(* IEC 61131-3 sources: SIMERLIFT/LOGICAD/SIMERLIFT/src_FBD/BCU, 6 files *)

(* ---- BatteryTypes.iecst ---- *)
TYPE
    BATTSTATE : USINT( STANDBY := 101,
    				  STARTUP := 102,
    				  PRECHARGE := 103,
    	              DISCHARGE := 104,
                      CHARGE := 105,
                      SHUTDOWN := 106,
                      FAULT := 107,
                      CHARGECOMPLETE := 108,
                      DISCHARGECOMPLETE := 109,
                      PRECHARGE4charge := 110);
END_TYPE

(* ---- ampMaxTempDis.iecst ---- *)
FUNCTION_BLOCK ampMultTempDis {
    width := 200;
  }

VAR_INPUT
temp:REAL;
END_VAR

VAR_OUTPUT
mult : REAL;
END_VAR

VAR
rstTimer:TON;
timeout:BOOL;
lastMult:REAL;
instantMult:REAL;
END_VAR

IF temp<-30 THEN
	mult:=0;
	instantMult:=0;
ELSIF temp<-25  THEN
	instantMult:=0.11;
ELSIF temp<-20  THEN
	instantMult:=0.15;
ELSIF temp<-15  THEN
	instantMult:=0.2;
ELSIF temp<-10  THEN
	instantMult:=0.25;
ELSIF temp<-5  THEN
	instantMult:=0.3;
ELSIF temp<0  THEN
	instantMult:=0.4;
ELSIF temp<5  THEN
	instantMult:=0.5;
ELSIF temp<10  THEN
	instantMult:=0.7;
ELSIF temp<50  THEN
	instantMult:=1;
ELSIF temp<55  THEN
	instantMult:=0.4;
ELSIF temp<56  THEN
	instantMult:=0.2;
ELSE
	mult:=0;
	instantMult:=0;
END_IF;

rstTimer(IN:=instantMult=lastMult, PT:=T#10s, Q=>timeout);

lastMult:=instantMult;

IF timeout THEN
	mult:=instantMult;
END_IF;

END_FUNCTION_BLOCK

(* ---- Arr2Val.iecst ---- *)
FUNCTION_BLOCK ARR2VAL  {
    width := 200;
  }

VAR_INPUT
	MaxBMU:USINT;
    indx:USINT;
	Map:ARRAY[0..15] OF USINT;
	CellCounter:USINT;
END_VAR

VAR_OUTPUT
	numofCell : UINT;
	Reset:BOOL;
END_VAR

Reset:=FALSE;
numofCell:=Map[indx];

IF (NOT Reset) AND (indx = MaxBMU - 1) AND (CellCounter = Map[indx]) THEN
    Reset := TRUE;
END_IF;

END_FUNCTION_BLOCK

(* ---- BCU_ID.iecfbd ---- *)
FUNCTION_BLOCK BCU_ID
  {
    height := 138;
    width := 290;
  }

  VAR
    TON1 : TON;
  END_VAR
  VAR_INPUT
    ADDR_BIT0 : BOOL;
    ADDR_BIT1 : BOOL;
    ADDR_BIT2 : BOOL;
  END_VAR
  VAR_OUTPUT
    PACK_ID : USINT;
    CAN_ID_10 : UDINT;
    CAN_ID_11 : UDINT;
    CAN_ID_12 : UDINT;
    CAN_ID_13 : UDINT;
    CAN_ID_14 : UDINT;
    CAN_ID_15 : UDINT;
    CAN_ID_16 : UDINT;
  END_VAR

  (*

    // Network 1:
    SEL(G := ADDR_BIT0, IN0 := 16#00, IN1 := 16#01, SEL => @C(10).SEL);
    SEL(G := ADDR_BIT1, IN0 := 16#00, IN1 := 16#02, SEL => @C(9).SEL);
    SEL(G := ADDR_BIT2, IN0 := 16#00, IN1 := 16#04, SEL => @C(11).SEL);
    ADD(IN1 := @C(10).SEL, IN2 := @C(9).SEL, IN3 := @C(11).SEL, ADD => PACK_ID);

    // Network 2:
    TON1(IN := 1, PT := T#1s);
    TO_UDINT(IN := TON1.Q, TO_UDINT => @C(36).TO_UDINT);
    ADD(IN1 := 16#18FF10F0, IN2 := PACK_ID, ADD => @C(26).ADD);
    MUL(IN1 := @C(36).TO_UDINT, IN2 := @C(26).ADD, MUL => CAN_ID_10);
    ADD(IN1 := 16#18FF11F0, IN2 := PACK_ID, ADD => @C(30).ADD);
    MUL(IN1 := @C(36).TO_UDINT, IN2 := @C(30).ADD, MUL => CAN_ID_11);
    ADD(IN1 := 16#18FF12F0, IN2 := PACK_ID, ADD => @C(38).ADD);
    MUL(IN1 := @C(36).TO_UDINT, IN2 := @C(38).ADD, MUL => CAN_ID_12);
    ADD(IN1 := 16#18FF13F0, IN2 := PACK_ID, ADD => @C(54).ADD);
    MUL(IN1 := @C(36).TO_UDINT, IN2 := @C(54).ADD, MUL => CAN_ID_13);
    ADD(IN1 := 16#18FF14F0, IN2 := PACK_ID, ADD => @C(25).ADD);
    MUL(IN1 := @C(36).TO_UDINT, IN2 := @C(25).ADD, MUL => CAN_ID_14);
    ADD(IN1 := 16#18FF15F0, IN2 := PACK_ID, ADD => @C(39).ADD);
    MUL(IN1 := @C(36).TO_UDINT, IN2 := @C(39).ADD, MUL => CAN_ID_15);
    ADD(IN1 := 16#18FF16F0, IN2 := PACK_ID, ADD => @C(67).ADD);
    MUL(IN1 := @C(36).TO_UDINT, IN2 := @C(67).ADD, MUL => CAN_ID_16);

  *)

  @VF(4) : @E(16#01), @R(330.0, 120.0, 90.0, 19.0), USINT;
  @C(7) : @F(ADD), @R(660.0, 120.0, 40.0, 58.0), USINT, @I(@N(IN1), @L(9.5)), @I(@N(IN2), @L(29.5)), @I(@N(IN3), @L(49.5)), @O(@N(ADD), @R(9.5));
  @C(10) : @F(SEL), @R(470.0, 80.0, 120.0, 58.0), USINT, @I(@N(G), @L(9.5)), @I(@N(IN0), @L(29.5)), @I(@N(IN1), @L(49.5)), @O(@N(SEL), @R(9.5));
  @C(9) : @F(SEL), @R(470.0, 140.0, 120.0, 58.0), USINT, @I(@N(G), @L(9.5)), @I(@N(IN0), @L(29.5)), @I(@N(IN1), @L(49.5)), @O(@N(SEL), @R(9.5));
  @C(11) : @F(SEL), @R(470.0, 200.0, 120.0, 58.0), USINT, @I(@N(G), @L(9.5)), @I(@N(IN0), @L(29.5)), @I(@N(IN1), @L(49.5)), @O(@N(SEL), @R(9.5));
  @VF(1) : @E(ADDR_BIT0), @R(90.0, 80.0, 140.0, 19.0);
  @VF(14) : @E(16#00), @R(330.0, 100.0, 90.0, 19.0), USINT;
  @VF(17) : @E(ADDR_BIT1), @R(90.0, 140.0, 140.0, 19.0);
  @VF(19) : @E(16#02), @R(330.0, 180.0, 90.0, 19.0), USINT;
  @VF(21) : @E(16#04), @R(330.0, 240.0, 90.0, 19.0), USINT;
  @VF(5) : @E(ADDR_BIT2), @R(90.0, 200.0, 140.0, 19.0);
  @VF(23) : @E(PACK_ID), @R(790.0, 120.0, 140.0, 19.0);
  @VF(468) : @E(16#18FF10F0), @R(280.0, 330.0, 220.0, 19.0), UDINT;
  @VF(33) : @E(CAN_ID_10), @R(790.0, 310.0, 140.0, 19.0);
  @C(41) : @F(MUL), @R(690.0, 310.0, 40.0, 38.0), UDINT, @I(@N(IN1), @L(9.5)), @I(@N(IN2), @L(29.5)), @O(@N(MUL), @R(9.5));
  @C(36) : @F(TO_UDINT), @R(290.0, 310.0, 120.0, 18.0), BOOL, @I(@N(IN), @L(9.5)), @O(@N(TO_UDINT), @R(9.5));
  @C(43) : @FB(TON1), @R(160.0, 310.0, 100.0, 38.0), @I(@N(IN), @L(9.5)), @I(@N(PT), @L(29.5)), @O(@N(Q), @R(9.5)), @O(@N(ET), @R(29.5));
  @VF(46) : @E(1), @R(70.0, 310.0, 70.0, 19.0), BOOL;
  @VF(48) : @E(T#1s), @R(70.0, 330.0, 70.0, 19.0);
  @C(51) : @F(MUL), @R(690.0, 350.0, 40.0, 38.0), UDINT, @I(@N(IN1), @L(9.5)), @I(@N(IN2), @L(29.5)), @O(@N(MUL), @R(9.5));
  @VF(58) : @E(CAN_ID_11), @R(790.0, 350.0, 140.0, 19.0);
  @C(59) : @F(MUL), @R(690.0, 390.0, 40.0, 38.0), UDINT, @I(@N(IN1), @L(9.5)), @I(@N(IN2), @L(29.5)), @O(@N(MUL), @R(9.5));
  @VF(73) : @E(CAN_ID_12), @R(790.0, 390.0, 140.0, 19.0);
  @C(83) : @F(MUL), @R(690.0, 430.0, 40.0, 38.0), UDINT, @I(@N(IN1), @L(9.5)), @I(@N(IN2), @L(29.5)), @O(@N(MUL), @R(9.5));
  @VF(88) : @E(CAN_ID_13), @R(790.0, 430.0, 140.0, 19.0);
  @C(98) : @F(MUL), @R(690.0, 470.0, 40.0, 38.0), UDINT, @I(@N(IN1), @L(9.5)), @I(@N(IN2), @L(29.5)), @O(@N(MUL), @R(9.5));
  @VF(103) : @E(CAN_ID_14), @R(790.0, 470.0, 140.0, 19.0);
  @C(113) : @F(MUL), @R(690.0, 510.0, 40.0, 38.0), UDINT, @I(@N(IN1), @L(9.5)), @I(@N(IN2), @L(29.5)), @O(@N(MUL), @R(9.5));
  @VF(118) : @E(CAN_ID_15), @R(790.0, 510.0, 140.0, 19.0);
  @C(26) : @F(ADD), @R(580.0, 330.0, 40.0, 38.0), UDINT, @I(@N(IN1), @L(9.5)), @I(@N(IN2), @L(29.5)), @O(@N(ADD), @R(9.5));
  @C(30) : @F(ADD), @R(580.0, 370.0, 40.0, 38.0), UDINT, @I(@N(IN1), @L(9.5)), @I(@N(IN2), @L(29.5)), @O(@N(ADD), @R(9.5));
  @VF(32) : @E(16#18FF11F0), @R(280.0, 370.0, 220.0, 19.0), UDINT;
  @C(38) : @F(ADD), @R(580.0, 410.0, 40.0, 38.0), UDINT, @I(@N(IN1), @L(9.5)), @I(@N(IN2), @L(29.5)), @O(@N(ADD), @R(9.5));
  @VF(40) : @E(16#18FF12F0), @R(280.0, 410.0, 220.0, 19.0), UDINT;
  @C(54) : @F(ADD), @R(580.0, 450.0, 40.0, 38.0), UDINT, @I(@N(IN1), @L(9.5)), @I(@N(IN2), @L(29.5)), @O(@N(ADD), @R(9.5));
  @VF(56) : @E(16#18FF13F0), @R(280.0, 450.0, 220.0, 19.0), UDINT;
  @C(25) : @F(ADD), @R(580.0, 490.0, 40.0, 38.0), UDINT, @I(@N(IN1), @L(9.5)), @I(@N(IN2), @L(29.5)), @O(@N(ADD), @R(9.5));
  @VF(28) : @E(16#18FF14F0), @R(280.0, 490.0, 220.0, 19.0), UDINT;
  @C(39) : @F(ADD), @R(580.0, 530.0, 40.0, 38.0), UDINT, @I(@N(IN1), @L(9.5)), @I(@N(IN2), @L(29.5)), @O(@N(ADD), @R(9.5));
  @VF(42) : @E(16#18FF15F0), @R(280.0, 530.0, 220.0, 19.0), UDINT;
  @VF(64) : @E(PACK_ID), @R(360.0, 350.0, 140.0, 19.0);
  @C(67) : @F(ADD), @R(580.0, 570.0, 40.0, 38.0), UDINT, @I(@N(IN1), @L(9.5)), @I(@N(IN2), @L(29.5)), @O(@N(ADD), @R(9.5));
  @VF(68) : @E(16#18FF16F0), @R(280.0, 570.0, 220.0, 19.0), UDINT;
  @C(70) : @F(MUL), @R(690.0, 550.0, 40.0, 38.0), UDINT, @I(@N(IN1), @L(9.5)), @I(@N(IN2), @L(29.5)), @O(@N(MUL), @R(9.5));
  @VF(72) : @E(CAN_ID_16), @R(790.0, 550.0, 140.0, 19.0);
  @CP(16) : 439.5, 109.5;
  @CP(53) : 659.5, 319.5;
  @CP(66) : 539.5, 359.5;

  @G(8) :
     @L(@C(10).SEL, @C(7).IN1)
    ;
  @G(12) :
     @L(@C(9).SEL, @C(7).IN2)
    ;
  @G(13) :
     @L(@C(11).SEL, @C(7).IN3)
    ;
  @G(2) :
     @L(@VF(1).o, @C(10).G)
    ;
  @G(3) :
     @L(@VF(4).o, @C(10).IN1)
    ;
  @G(15) :
     @L(@VF(14).o, @CP(16)),
     @L(@CP(16), @C(10).IN0),
     @L(@CP(16), @C(9).IN0),
     @L(@CP(16), @C(11).IN0)
    ;
  @G(18) :
     @L(@VF(17).o, @C(9).G)
    ;
  @G(20) :
     @L(@VF(19).o, @C(9).IN1)
    ;
  @G(22) :
     @L(@VF(21).o, @C(11).IN1)
    ;
  @G(6) :
     @L(@VF(5).o, @C(11).G)
    ;
  @G(24) :
     @L(@C(7).ADD, @VF(23).i)
    ;
  @G(44) :
     @L(@C(43).Q, @C(36).IN)
    ;
  @G(45) :
     @L(@C(36).TO_UDINT, @CP(53)),
     @L(@CP(53), @C(41).IN1),
     @L(@CP(53), @C(51).IN1),
     @L(@CP(53), @C(59).IN1),
     @L(@CP(53), @C(83).IN1),
     @L(@CP(53), @C(98).IN1),
     @L(@CP(53), @C(113).IN1),
     @L(@CP(53), @C(70).IN1)
    ;
  @G(47) :
     @L(@VF(46).o, @C(43).IN)
    ;
  @G(49) :
     @L(@VF(48).o, @C(43).PT)
    ;
  @G(50) :
     @L(@C(41).MUL, @VF(33).i)
    ;
  @G(63) :
     @L(@C(51).MUL, @VF(58).i)
    ;
  @G(76) :
     @L(@C(59).MUL, @VF(73).i)
    ;
  @G(91) :
     @L(@C(83).MUL, @VF(88).i)
    ;
  @G(106) :
     @L(@C(98).MUL, @VF(103).i)
    ;
  @G(121) :
     @L(@C(113).MUL, @VF(118).i)
    ;
  @G(27) :
     @L(@VF(468).o, @C(26).IN1)
    ;
  @G(29) :
     @L(@C(26).ADD, @C(41).IN2)
    ;
  @G(35) :
     @L(@VF(32).o, @C(30).IN1)
    ;
  @G(37) :
     @L(@C(30).ADD, @C(51).IN2)
    ;
  @G(52) :
     @L(@VF(40).o, @C(38).IN1)
    ;
  @G(60) :
     @L(@VF(56).o, @C(54).IN1)
    ;
  @G(31) :
     @L(@VF(28).o, @C(25).IN1)
    ;
  @G(34) :
     @L(@C(25).ADD, @C(98).IN2)
    ;
  @G(55) :
     @L(@VF(42).o, @C(39).IN1)
    ;
  @G(57) :
     @L(@C(39).ADD, @C(113).IN2)
    ;
  @G(61) :
     @L(@C(54).ADD, @C(83).IN2)
    ;
  @G(62) :
     @L(@C(38).ADD, @C(59).IN2)
    ;
  @G(65) :
     @L(@VF(64).o, @CP(66)),
     @L(@CP(66), @C(26).IN2),
     @L(@CP(66), @C(30).IN2),
     @L(@CP(66), @C(38).IN2),
     @L(@CP(66), @C(54).IN2),
     @L(@CP(66), @C(25).IN2),
     @L(@CP(66), @C(39).IN2),
     @L(@CP(66), @C(67).IN2)
    ;
  @G(69) :
     @L(@VF(68).o, @C(67).IN1)
    ;
  @G(71) :
     @L(@C(67).ADD, @C(70).IN2)
    ;
  @G(74) :
     @L(@C(70).MUL, @VF(72).i)
    ;
END_FUNCTION_BLOCK

(* ---- essState1.iecst ---- *)
FUNCTION_BLOCK  essState1  {
    fault {index := 12};
    shutdownComplete {index := 11};
    chargeProtect {index := 9};
    dischargeProtect {index := 8};
    contactFbkNeg {loc := "left", index := 6};
    contactFbk {loc := "left", index := 5};
    prechargeOk {loc := "left", index := 4};
    contactNeg {loc := "right", index := 4};
    contact {loc := "right", index := 3};
    prechargeOn {loc := "right", index := 2};
    width := 400;
    bgColor := "mediumseagreen";
    height := 258;
  }

VAR_INPUT
	discharge:BOOL;
	charge:BOOL;
	shutdown:BOOL;

	prechargeOk:BOOL;
	contactFbk:BOOL;
	contactFbkNeg:BOOL;

	dischargeProtect:BOOL;
	chargeProtect:BOOL;

	shutdownComplete:BOOL;
	fault:BOOL;
END_VAR

VAR_OUTPUT
	STATE : BATTSTATE;

	prechargeOn:BOOL;
	contact:BOOL;
	contactNeg:BOOL;
END_VAR

VAR

BATTERYSTATE:BATTSTATE:=BATTSTATE#STANDBY;
PREVSTATE:BATTSTATE:=BATTSTATE#STANDBY;

BATTIMER:TON;
BATSTATEINTERVAL:TIME:=T#10s;
BATSTATETIMEOUT:BOOL;
BATSTATEELAPSEDTIME:TIME;
STANDBYINTERVAL:TIME:=T#2s;
FaultCounter: USINT;

contactFbkTimer : TON;
END_VAR

BATTIMER(IN:=BATTERYSTATE=PREVSTATE, PT:=BATSTATEINTERVAL, Q=>BATSTATETIMEOUT, ET=>BATSTATEELAPSEDTIME);

PREVSTATE:=BATTERYSTATE;

CASE BATTERYSTATE OF

	BATTSTATE#STANDBY:  // standby
		STATE:=BATTSTATE#STANDBY;
		BATSTATEINTERVAL:=T#12s;
		FaultCounter := 0;
		contact:=0;
		contactNeg:=0;

        IF BATSTATEELAPSEDTIME>STANDBYINTERVAL THEN
        	STANDBYINTERVAL:=T#500ms;
        	IF fault THEN
				BATTERYSTATE:=BATTSTATE#FAULT;
			ELSIF shutdown THEN
				BATTERYSTATE:=BATTSTATE#SHUTDOWN;
			ELSIF discharge THEN
				IF prechargeOk THEN
					BATTERYSTATE:=BATTSTATE#DISCHARGE;
				ELSE
					BATTERYSTATE:=BATTSTATE#PRECHARGE;
				END_IF;
			ELSIF charge THEN
				BATTERYSTATE:=BATTSTATE#CHARGE;
			END_IF;
        END_IF;

	BATTSTATE#PRECHARGE:
		IF prechargeOk AND discharge THEN
			BATTERYSTATE := BATTSTATE#DISCHARGE;
		ELSIF discharge AND NOT prechargeOk THEN
			STATE := BATTSTATE#PRECHARGE;
			//BATSTATEINTERVAL:=T#5s;
			contact := 0;
			contactNeg := 0;
			prechargeOn := discharge;
			FaultCounter:=0;

			contactFbkTimer(IN := TRUE, PT := T#5s);
			IF contactFbkTimer.Q THEN
				IF fault OR shutdown OR BATSTATETIMEOUT THEN
					BATTERYSTATE := BATTSTATE#SHUTDOWN;
				ELSE
					BATTERYSTATE := BATTSTATE#DISCHARGE;
				END_IF;
			END_IF;
		ELSE
			BATTERYSTATE := BATTSTATE#SHUTDOWN;
		END_IF;

	BATTSTATE#DISCHARGE:  //discharge
		STATE:=BATTSTATE#DISCHARGE;
		BATSTATEINTERVAL:=T#120s;

		prechargeOn:=1;
		contact:=0;
		contactNeg:=1;

		IF discharge THEN
			contactFbkTimer(IN := NOT contactFbkNeg, PT := T#5s);
			IF contactFbkTimer.Q THEN
				IF fault OR shutdown OR NOT contactFbkNeg THEN
					IF FaultCounter<2 THEN
						FaultCounter:=Faultcounter+1;
					ELSE
						BATTERYSTATE:=BATTSTATE#SHUTDOWN;
					END_IF;
				ELSE
					FaultCounter:=0;
				END_IF;
			END_IF;
		ELSIF charge AND NOT chargeProtect THEN
			BATTERYSTATE:=BATTSTATE#CHARGE;
		ELSE
			BATTERYSTATE:=BATTSTATE#SHUTDOWN;
		END_IF;
		contactFbkTimer(IN := FALSE);

	BATTSTATE#CHARGE:  // charge
		STATE:=BATTSTATE#CHARGE;
		BATSTATEINTERVAL:=T#120s;

		prechargeOn:=0;
		contact:=1;
		contactNeg:=0;
		FaultCounter:=0;

		IF charge THEN
			contactFbkTimer(IN := NOT contactFbk, PT := T#2s);
			IF contactFbkTimer.Q THEN
				IF fault OR shutdown OR NOT contactFbk THEN
					BATTERYSTATE:=BATTSTATE#SHUTDOWN;
				ELSIF NOT charge THEN
					IF discharge THEN
						BATTERYSTATE:=BATTSTATE#PRECHARGE;
					ELSE
						BATTERYSTATE:=BATTSTATE#SHUTDOWN;
					END_IF;
				END_IF;
			END_IF;
		ELSIF discharge THEN
			BATTERYSTATE:=BATTSTATE#PRECHARGE;
		ELSE
			BATTERYSTATE:=BATTSTATE#SHUTDOWN;
		END_IF;
		contactFbkTimer(IN := FALSE);

	BATTSTATE#SHUTDOWN:  // shutdown
		STATE:=BATTSTATE#SHUTDOWN;
		BATSTATEINTERVAL:=T#5000ms;

		prechargeOn:=0;
		FaultCounter:=0;

		IF shutdown OR BATSTATEELAPSEDTIME>T#2000ms OR (shutdownComplete AND (BATSTATEELAPSEDTIME>T#500ms))  THEN
			contact:=0;
			contactNeg:=0;
			IF fault THEN
				BATTERYSTATE:=BATTSTATE#FAULT;
			ELSIF shutdown THEN
				BATTERYSTATE:=BATTSTATE#SHUTDOWN;
			ELSIF NOT contactFbk AND NOT contactFbkNeg THEN
				IF dischargeProtect THEN
					BATTERYSTATE:=BATTSTATE#DISCHARGECOMPLETE;
				ELSIF chargeProtect THEN
					BATTERYSTATE:=BATTSTATE#CHARGECOMPLETE;
				ELSIF BATSTATETIMEOUT OR charge OR discharge THEN
					BATTERYSTATE:=BATTSTATE#STANDBY;
				END_IF;
			END_IF;
		END_IF;

	BATTSTATE#FAULT:  //fault
		STATE:=BATTSTATE#FAULT;
		BATSTATEINTERVAL:=T#10s;

		contact:=0;
		contactNeg:=0;
		prechargeOn:=0;
		FaultCounter:=0;

		IF NOT fault AND BATSTATETIMEOUT THEN
			BATTERYSTATE:=BATTSTATE#SHUTDOWN;
		END_IF;

	BATTSTATE#CHARGECOMPLETE:
		STATE:=BATTSTATE#CHARGECOMPLETE;
		BATSTATEINTERVAL:=T#5s;

		prechargeOn:=0;
		contact:=0;
		contactNeg:=0;
		FaultCounter:=0;

		IF fault THEN
			BATTERYSTATE:=BATTSTATE#FAULT;
		ELSIF shutdown THEN
			BATTERYSTATE:=BATTSTATE#SHUTDOWN;
		ELSIF BATSTATETIMEOUT AND discharge THEN
			BATTERYSTATE:=BATTSTATE#STANDBY;
		END_IF;

	BATTSTATE#DISCHARGECOMPLETE:
		STATE:=BATTSTATE#DISCHARGECOMPLETE;
		BATSTATEINTERVAL:=T#5s;

		prechargeOn:=0;
		contact:=0;
		contactNeg:=0;
		FaultCounter:=0;

		IF fault THEN
			BATTERYSTATE:=BATTSTATE#FAULT;
		ELSIF shutdown THEN
			BATTERYSTATE:=BATTSTATE#SHUTDOWN;
		ELSIF BATSTATETIMEOUT AND charge THEN
			BATTERYSTATE:=BATTSTATE#STANDBY;
		END_IF;

END_CASE;

END_FUNCTION_BLOCK

(* ---- numOfCells.iecst ---- *)
FUNCTION_BLOCK numOfCells  {
    width := 300;
  }

VAR_INPUT
    numofBMU:USINT;
	cellMap:ARRAY[0..15] OF USINT;
END_VAR

VAR_OUTPUT
	numofCell : UINT;
END_VAR

VAR
i:USINT;

END_VAR

numofCell:=0;

FOR i:=1 TO numofBMU By 1 DO
	numofCell:=numofCell+cellMap[i-1];
END_FOR;

END_FUNCTION_BLOCK
